// TwinCAT 3 PLC project SequentialTestSuitesAndTests
// Title: TcUnit sequentially running tests example projects
// Company: www.tcunit.org
// Author: Jakob Sagatowski
// ProjectVersion: 1.0.0.0
// ProgramVersion: 3.1.4022.7
// libraries:
//   Tc2_EtherCAT, * (Beckhoff Automation GmbH)
//   Tc2_Standard, * (Beckhoff Automation GmbH)
//   Tc2_System, * (Beckhoff Automation GmbH)
//   Tc3_Module, * (Beckhoff Automation GmbH)
//   TcUnit, * (www.tcunit.org)
// project tree:
//   DUTs/ E_DIAGNOSISTYPE.TcDUT, E_DIAGNOSTICCODETYPE.TcDUT, E_EVENTQUALIFIERMODE.TcDUT, E_TIMESTAMPTYPE.TcDUT (not stored), ST_DIAGNOSTICCODE.TcDUT (not stored), ST_DIAGNOSTICMESSAGE.TcDUT (not stored), ST_FLAGS.TcDUT (not stored)
//   GVLs/ GVL.TcGVL
//   / PlcTask.TcTTO
//   POUs/ FB_DiagnosticMessageDiagnosticCodeParser.TcPOU, FB_DiagnosticMessageFlagsParser.TcPOU, FB_DiagnosticMessageParser.TcPOU, FB_DiagnosticMessageTextIdentityParser.TcPOU, FB_DiagnosticMessageTimeStampParser.TcPOU, F_DWORDFromBytes.TcPOU (not stored), F_WORDFromBytes.TcPOU
//   Test/ FB_DiagnosticMessageDiagnosticCodeParser_Test.TcPOU, FB_DiagnosticMessageFlagsParser_Test.TcPOU, FB_DiagnosticMessageParser_Test.TcPOU, FB_DiagnosticMessageTextIdentityParser_Test.TcPOU, FB_DiagnosticMessageTimeStampParser_Test.TcPOU, PRG_TEST.TcPOU
// real-time tasks:
//   TASK PlcTask: cycle T#10ms, priority 20, ADS port 350

CONFIGURATION SequentialTestSuitesAndTests
    RESOURCE PLC ON TwinCAT3
        TASK PlcTask(INTERVAL := T#10ms, PRIORITY := 20);
        PROGRAM PRG_TEST WITH PlcTask : PRG_TEST;
    END_RESOURCE
END_CONFIGURATION

// ---- DUTs/E_DIAGNOSISTYPE.TcDUT
{attribute 'qualified_only'}
TYPE E_DIAGNOSISTYPE :
(
    InfoMessage := 0,
    WarningMessage := 1,
    ErrorMessage := 2,
    Unspecified := 3
) BYTE;
END_TYPE

// ---- DUTs/E_DIAGNOSTICCODETYPE.TcDUT
{attribute 'qualified_only'}
{attribute 'strict'}
TYPE E_DIAGNOSTICCODETYPE :
(
    ManufacturerSpecific := 0,
    EmergencyErrorCodeDS301 := 1,
    ProfileSpecific := 2,
    Unspecified := 3
) USINT;
END_TYPE

// ---- DUTs/E_EVENTQUALIFIERMODE.TcDUT
{attribute 'qualified_only'}
TYPE E_EVENTQUALIFIERMODE :
(
	Reserved := 0,
    EventSingleShot := 1,
    EventDisappears := 2,
    EventAppears := 3
) USINT;
END_TYPE

// ---- GVLs/GVL.TcGVL
{attribute 'qualified_only'}
VAR_GLOBAL
    fbDiagnosticMessageDiagnosticCodeParser_Test_WhenEmergencyErrorCodeExpectEmergencyErrorCode : ULINT;
    fbDiagnosticMessageDiagnosticCodeParser_Test_WhenManufacturerSpecificExpectManufacturerSpecific : ULINT;
    fbDiagnosticMessageDiagnosticCodeParser_Test_WhenProfileSpecificExpectProfileSpecific : ULINT;
    fbDiagnosticMessageDiagnosticCodeParser_Test_WhenReservedForFutureUseExpectReservedForFutureUse : ULINT;

    fbDiagnosticMessageFlagsParser_Test_WhenInfoMessageExpectInfoMessageGlobalTimestampAndZeroParameters : ULINT;
    fbDiagnosticMessageFlagsParser_Test_WhenWarningMessageExpectWarningMessageLocalTimestampAndTwoParameters : ULINT;
    fbDiagnosticMessageFlagsParser_Test_WhenErrorMessageExpectErrorMessageLocalTimestampAndFourParameters : ULINT;
    fbDiagnosticMessageFlagsParser_Test_WhenReservedForFutureUseMessageExpectReservedForFutureUseMessageLocalTimestampAnd33Parameters : ULINT;    

    fbDiagnosticMessageParser_Test_TestWithEmergencyMessage : ULINT;
    fbDiagnosticMessageParser_Test_TestWithManufacturerSpecificMessage : ULINT;
    fbDiagnosticMessageParser_Test_TestWithUnspecifiedMessageMessage : ULINT;
    fbDiagnosticMessageParser_Test_TestWithUnspecifiedMessageMessage_ParameterVariant : ULINT;

    fbDiagnosticMessageTextIdentityParser_Test_WhenTextIdentityLowExpectTextIdentity0 : ULINT;
    fbDiagnosticMessageTextIdentityParser_Test_WhenTextIdentityHighExpectTextIdentity65535 : ULINT;
    fbDiagnosticMessageTextIdentityParser_Test_WhenTextIdentityMedExpectTextIdentity34500 : ULINT;

    fbDiagnosticMessageTimeStampParser_Test_TestWithTimestampZeroTimeExpectCurrentTime : ULINT;
    fbDiagnosticMessageTimeStampParser_Test_TestWithValidTimestampExpectSameTimestamp : ULINT;
END_VAR

// ---- Test/PRG_TEST.TcPOU
(*
    This is the main program for execution of the unit tests.
    The program executes the test suites one after the other, with a delay of T#0MS between
    each other (that is, as soon as one test suite has finished executing, the next
    one starts to execute immediately after). This delay is defined in the parameter
    GVL_Param_TcUnit.TimeBetweenTestSuitesExecution (default T#0MS).
    Within each test suite, the program also executes each test one after the other, which
    is achieved by calling the TEST_ORDERED() for every test. The test-order is defined
    by the order of which the tests are being called.
*)
PROGRAM PRG_TEST
VAR
    (* Test function blocks *)
    fbDiagnosticMessageDiagnosticCodeParser_Test : FB_DiagnosticMessageDiagnosticCodeParser_Test;
    fbDiagnosticMessageFlagsParser_Test : FB_DiagnosticMessageFlagsParser_Test;
    fbDiagnosticMessageParser_Test : FB_DiagnosticMessageParser_Test;
    fbDiagnosticMessageTextIdentityParser_Test : FB_DiagnosticMessageTextIdentityParser_Test;
    fbDiagnosticMessageTimeStampParser_Test : FB_DiagnosticMessageTimeStampParser_Test;
END_VAR

TcUnit.RUN_IN_SEQUENCE();

END_PROGRAM

// ---- Test/FB_DiagnosticMessageDiagnosticCodeParser_Test.TcPOU
FUNCTION_BLOCK FB_DiagnosticMessageDiagnosticCodeParser_Test EXTENDS TcUnit.FB_TestSuite

(* The tests are run in the order that they are called. Asserts are not evaluated before the previous test has called TEST_FINISHED() *)
WhenEmergencyErrorCodeExpectEmergencyErrorCode();
WhenManufacturerSpecificExpectManufacturerSpecific();
WhenProfileSpecificExpectProfileSpecific();
WhenReservedForFutureUseExpectReservedForFutureUse();

METHOD PRIVATE WhenEmergencyErrorCodeExpectEmergencyErrorCode
VAR
    fbDiagnosticMessageDiagnosticCodeParser : FB_DiagnosticMessageDiagnosticCodeParser;
    stDiagnosticCode : ST_DIAGNOSTICCODE;
END_VAR
VAR CONSTANT
    // @TEST-FIXTURE EmergencyErrorCode
    cnDiagnosticCodeBufferByte1_EmergencyErrorCode : BYTE := 16#00; // 16#E800
    cnDiagnosticCodeBufferByte2_EmergencyErrorCode : BYTE := 16#E8;
    cnDiagnosticCodeBufferByte3_EmergencyErrorCode : BYTE := 16#30; // 16#7530 = 10#30000
    cnDiagnosticCodeBufferByte4_EmergencyErrorCode : BYTE := 16#75;
    canDiagnosticCodeBuffer_EmergencyErrorCode : ARRAY[1..4] OF BYTE := [
                                                cnDiagnosticCodeBufferByte1_EmergencyErrorCode,
                                                cnDiagnosticCodeBufferByte2_EmergencyErrorCode,
                                                cnDiagnosticCodeBufferByte3_EmergencyErrorCode,
                                                cnDiagnosticCodeBufferByte4_EmergencyErrorCode];
    // @TEST-RESULT EmergencyErrorCode
    ceDiagnosticCodeType_EmergencyErrorCode : E_DIAGNOSTICCODETYPE := E_DIAGNOSTICCODETYPE.EmergencyErrorCodeDS301;
    cnDiagnosticCode_EmergencyErrorCode : UINT := 10#30000;
END_VAR
IF TEST_ORDERED('WhenEmergencyErrorCodeExpectEmergencyErrorCode') THEN
    GVL.fbDiagnosticMessageDiagnosticCodeParser_Test_WhenEmergencyErrorCodeExpectEmergencyErrorCode := GVL.fbDiagnosticMessageDiagnosticCodeParser_Test_WhenEmergencyErrorCodeExpectEmergencyErrorCode + 1; // Only for testing the framework. Ignore this.
    // @TEST-RUN
    fbDiagnosticMessageDiagnosticCodeParser(anDiagnosticCodeBuffer := canDiagnosticCodeBuffer_EmergencyErrorCode,
                                            stDiagnosticCode => stDiagnosticCode);

    // @TEST-ASSERT
    AssertEquals_USINT(Expected := ceDiagnosticCodeType_EmergencyErrorCode,
                       Actual := stDiagnosticCode.eDiagnosticCodeType,
                       Message := 'Test $'emergency error code$' failed at $'diagnostic code type$'');
    AssertEquals_UINT(Expected := cnDiagnosticCode_EmergencyErrorCode,
                      Actual := stDiagnosticCode.nCode,
                      Message := 'Test $'emergency error code$' failed at $'diagnostic code$'');
    TEST_FINISHED();
END_IF
END_METHOD

METHOD PRIVATE WhenManufacturerSpecificExpectManufacturerSpecific
VAR
    fbDiagnosticMessageDiagnosticCodeParser : FB_DiagnosticMessageDiagnosticCodeParser;
    stDiagnosticCode : ST_DIAGNOSTICCODE;
END_VAR
VAR CONSTANT
    // @TEST-FIXTURE ManuFacturerSpecific
    cnDiagnosticCodeBufferByte1_ManufacturerSpecific : BYTE := 16#00; // 16#E000 (in range of 0xE000 - 0xE7FF)
    cnDiagnosticCodeBufferByte2_ManufacturerSpecific : BYTE := 16#E0;
    cnDiagnosticCodeBufferByte3_ManufacturerSpecific : BYTE := 16#E8; // 16#03E8 = 10#1000
    cnDiagnosticCodeBufferByte4_ManufacturerSpecific : BYTE := 16#03;
    canDiagnosticCodeBuffer_ManufacturerSpecific : ARRAY[1..4] OF BYTE := [
                                                cnDiagnosticCodeBufferByte1_ManufacturerSpecific,
                                                cnDiagnosticCodeBufferByte2_ManufacturerSpecific,
                                                cnDiagnosticCodeBufferByte3_ManufacturerSpecific,
                                                cnDiagnosticCodeBufferByte4_ManufacturerSpecific];
                                                
    // @TEST-RESULT ManuFacturerSpecific
    ceDiagnosticCodeType_ManufacturerSpecific : E_DIAGNOSTICCODETYPE := E_DIAGNOSTICCODETYPE.ManufacturerSpecific;
    cnDiagnosticCode_ManufacturerSpecific : UINT := 10#1000;
END_VAR
IF TEST_ORDERED('WhenManufacturerSpecificExpectManufacturerSpecific') THEN
    GVL.fbDiagnosticMessageDiagnosticCodeParser_Test_WhenManufacturerSpecificExpectManufacturerSpecific := GVL.fbDiagnosticMessageDiagnosticCodeParser_Test_WhenManufacturerSpecificExpectManufacturerSpecific + 1; // Only for testing the framework. Ignore this.
    // @TEST-RUN
    fbDiagnosticMessageDiagnosticCodeParser(anDiagnosticCodeBuffer := canDiagnosticCodeBuffer_ManufacturerSpecific,
                                            stDiagnosticCode => stDiagnosticCode);

    // @TEST-ASSERT
    AssertEquals_USINT(Expected := ceDiagnosticCodeType_ManufacturerSpecific,
                       Actual := stDiagnosticCode.eDiagnosticCodeType,
                       Message := 'Test $'manufacturer specific$' failed at $'diagnostic code type$'');
    AssertEquals_UINT(Expected := cnDiagnosticCode_ManufacturerSpecific,
                      Actual := stDiagnosticCode.nCode,
                      Message := 'Test $'manufacturer specific$' failed at $'diagnostic code$'');

    TEST_FINISHED();
END_IF
END_METHOD

METHOD PRIVATE WhenProfileSpecificExpectProfileSpecific
VAR
    fbDiagnosticMessageDiagnosticCodeParser : FB_DiagnosticMessageDiagnosticCodeParser;
    stDiagnosticCode : ST_DIAGNOSTICCODE;
END_VAR
VAR CONSTANT
    // @TEST-FIXTURE ProfileSpecific
    cnDiagnosticCodeBufferByte1_ProfileSpecific : BYTE := 16#10; // 16#EF10 (in range of 0xEE00 - 0xEFFF)
    cnDiagnosticCodeBufferByte2_ProfileSpecific : BYTE := 16#EF;
    cnDiagnosticCodeBufferByte3_ProfileSpecific : BYTE := 16#FF; // 16#FFFF = 10#65535
    cnDiagnosticCodeBufferByte4_ProfileSpecific : BYTE := 16#FF;
    canDiagnosticCodeBuffer_ProfileSpecific : ARRAY[1..4] OF BYTE := [
                                                cnDiagnosticCodeBufferByte1_ProfileSpecific,
                                                cnDiagnosticCodeBufferByte2_ProfileSpecific,
                                                cnDiagnosticCodeBufferByte3_ProfileSpecific,
                                                cnDiagnosticCodeBufferByte4_ProfileSpecific];

    // @TEST-RESULT ProfileSpecific
    ceDiagnosticCodeType_ProfileSpecific : E_DIAGNOSTICCODETYPE := E_DIAGNOSTICCODETYPE.ProfileSpecific;
    cnDiagnosticCode_ProfileSpecific : UINT := 10#65535;
END_VAR
IF TEST_ORDERED('WhenProfileSpecificExpectProfileSpecific') THEN
    GVL.fbDiagnosticMessageDiagnosticCodeParser_Test_WhenProfileSpecificExpectProfileSpecific := GVL.fbDiagnosticMessageDiagnosticCodeParser_Test_WhenProfileSpecificExpectProfileSpecific + 1; // Only for testing the framework. Ignore this.
    // @TEST-RUN
    fbDiagnosticMessageDiagnosticCodeParser(anDiagnosticCodeBuffer := canDiagnosticCodeBuffer_ProfileSpecific,
                                            stDiagnosticCode => stDiagnosticCode);

    // @TEST-ASSERT
    AssertEquals_USINT(Expected := ceDiagnosticCodeType_ProfileSpecific,
                       Actual := stDiagnosticCode.eDiagnosticCodeType,
                       Message := 'Test $'profile specific$' failed at $'diagnostic code type$'');
    AssertEquals_UINT(Expected := cnDiagnosticCode_ProfileSpecific,
                      Actual := stDiagnosticCode.nCode,
                      Message := 'Test $'profile specific$' failed at $'diagnostic code$'');

    TEST_FINISHED();
END_IF
END_METHOD

METHOD PRIVATE WhenReservedForFutureUseExpectReservedForFutureUse
VAR
    fbDiagnosticMessageDiagnosticCodeParser : FB_DiagnosticMessageDiagnosticCodeParser;
    stDiagnosticCode : ST_DIAGNOSTICCODE;
END_VAR
VAR CONSTANT
    // @TEST-FIXTURE ReservedForFutureUse
    cnDiagnosticCodeBufferByte1_ReservedForFutureUse : BYTE := 16#01; // 16#E801 (in range of 0xE801 - 0xEDFF)
    cnDiagnosticCodeBufferByte2_ReservedForFutureUse : BYTE := 16#E8;
    cnDiagnosticCodeBufferByte3_ReservedForFutureUse : BYTE := 16#D9; // 16#3BD9 = 10#15321
    cnDiagnosticCodeBufferByte4_ReservedForFutureUse : BYTE := 16#3B;
    canDiagnosticCodeBuffer_ReservedForFutureUse : ARRAY[1..4] OF BYTE := [
                                                cnDiagnosticCodeBufferByte1_ReservedForFutureUse,
                                                cnDiagnosticCodeBufferByte2_ReservedForFutureUse,
                                                cnDiagnosticCodeBufferByte3_ReservedForFutureUse,
                                                cnDiagnosticCodeBufferByte4_ReservedForFutureUse];

    // @TEST-RESULT ReservedForFutureUse
    ceDiagnosticCodeType_ReservedForFutureUse : E_DIAGNOSTICCODETYPE := E_DIAGNOSTICCODETYPE.Unspecified;
    cnDiagnosticCode_ReservedForFutureUse : UINT := 10#15321;
END_VAR
IF TEST_ORDERED('WhenReservedForFutureUseExpectReservedForFutureUse') THEN
    GVL.fbDiagnosticMessageDiagnosticCodeParser_Test_WhenReservedForFutureUseExpectReservedForFutureUse := GVL.fbDiagnosticMessageDiagnosticCodeParser_Test_WhenReservedForFutureUseExpectReservedForFutureUse + 1; // Only for testing the framework. Ignore this.

    // @TEST-RUN
    fbDiagnosticMessageDiagnosticCodeParser(anDiagnosticCodeBuffer := canDiagnosticCodeBuffer_ReservedForFutureUse,
                                            stDiagnosticCode => stDiagnosticCode);

    // @TEST-ASSERT
    AssertEquals_USINT(Expected := ceDiagnosticCodeType_ReservedForFutureUse,
                       Actual := stDiagnosticCode.eDiagnosticCodeType,
                       Message := 'Test $'reserved for future use$' failed at $'diagnostic code type$'');
    AssertEquals_UINT(Expected := cnDiagnosticCode_ReservedForFutureUse,
                      Actual := stDiagnosticCode.nCode,
                      Message := 'Test $'reserved for future use$' failed at $'diagnostic code$'');

    TEST_FINISHED();
END_IF
END_METHOD

END_FUNCTION_BLOCK

// ---- POUs/FB_DiagnosticMessageDiagnosticCodeParser.TcPOU
(*
    This function block parses a the part "diagnostic code" of the diagnostic message according to the
    ETG.1020 protocol enhancements.
*)
FUNCTION_BLOCK FB_DiagnosticMessageDiagnosticCodeParser
VAR_INPUT
    anDiagnosticCodeBuffer : ARRAY[1..4] OF BYTE;
END_VAR
VAR_OUTPUT
    stDiagnosticCode : ST_DIAGNOSTICCODE;
END_VAR
VAR
    nDiagnosisCodeType : WORD;
    nDiagnosisCodeTypeLow : WORD;
    nCode : WORD;
    nCodeLow : WORD;
END_VAR
VAR CONSTANT
    cnNotUsedOne_Low : WORD := 16#0000;
    cnNotUsedOne_High : WORD := 16#DFFF;
    cnManufacturerSpecific_Low : WORD := 16#E000;
    cnManufacturerSpecific_High : WORD := 16#E7FF;
    cnEmergencyErrorCodeDS301 : WORD := 16#E800;
    cnReservedForFutureStandardization_Low : WORD := 16#E801;
    cnReservedForFutureStandardization_High : WORD := 16#EDFF;
    cnProfileSpecific_Low : WORD := 16#EE00;
    cnProfileSpecific_High : WORD := 16#EFFF;
    cnNotUsedTwo_Low : WORD := 16#F000;
    cnNotUsedTwo_High : WORD := 16#FFFF;
END_VAR

nDiagnosisCodeType := BYTE_TO_WORD(anDiagnosticCodeBuffer[2]);
nDiagnosisCodeType := SHL(nDiagnosisCodeType, 8);
nDiagnosisCodeTypeLow := BYTE_TO_WORD(anDiagnosticCodeBuffer[1]);
nDiagnosisCodeType := nDiagnosisCodeType OR nDiagnosisCodeTypeLow;

IF (nDiagnosisCodeType >= cnNotUsedOne_Low AND nDiagnosisCodeType <= cnNotUsedOne_High) OR
   (nDiagnosisCodeType >= cnReservedForFutureStandardization_Low AND
    nDiagnosisCodeType <= cnReservedForFutureStandardization_High) OR
   (nDiagnosisCodeType >= cnNotUsedTwo_Low AND nDiagnosisCodeType <= cnNotUsedTwo_High) THEN
   stDiagnosticCode.eDiagnosticCodeType := E_DIAGNOSTICCODETYPE.Unspecified;
ELSIF nDiagnosisCodeType >= cnManufacturerSpecific_Low AND nDiagnosisCodeType <= cnManufacturerSpecific_High THEN
    stDiagnosticCode.eDiagnosticCodeType := E_DIAGNOSTICCODETYPE.ManufacturerSpecific;
ELSIF nDiagnosisCodeType = cnEmergencyErrorCodeDS301 THEN
    stDiagnosticCode.eDiagnosticCodeType := E_DIAGNOSTICCODETYPE.EmergencyErrorCodeDS301;
ELSIF nDiagnosisCodeType >= cnProfileSpecific_Low AND nDiagnosisCodeType <= cnProfileSpecific_High THEN
    stDiagnosticCode.eDiagnosticCodeType := E_DIAGNOSTICCODETYPE.ProfileSpecific;
END_IF

nCode := BYTE_TO_WORD(anDiagnosticCodeBuffer[4]);
nCode := SHL(nCode, 8);
nCodeLow := BYTE_TO_WORD(anDiagnosticCodeBuffer[3]);
nCode := nCode OR nCodeLow;

stDiagnosticCode.nCode := WORD_TO_UINT(nCode);

END_FUNCTION_BLOCK

// ---- Test/FB_DiagnosticMessageFlagsParser_Test.TcPOU
FUNCTION_BLOCK FB_DiagnosticMessageFlagsParser_Test EXTENDS TcUnit.FB_TestSuite

(* The tests are run in the order that they are called. Asserts are not evaluated before the previous test has called TEST_FINISHED() *)
WhenInfoMessageExpectInfoMessageGlobalTimestampAndZeroParameters();
WhenWarningMessageExpectWarningMessageLocalTimestampAndTwoParameters();
WhenErrorMessageExpectErrorMessageLocalTimestampAndFourParameters();
WhenReservedForFutureUseMessageExpectReservedForFutureUseMessageLocalTimestampAnd33Parameters();

METHOD PRIVATE WhenErrorMessageExpectErrorMessageLocalTimestampAndFourParameters
VAR
    fbDiagnosticMessageFlagsParser : FB_DiagnosticMessageFlagsParser;
    stFlags : ST_FLAGS;

    // @TEST-FIXTURE ErrorMessage
    cnFlagsBufferByte1_ErrorMessage : BYTE := 2#0001_0010; // Error message and local time stamp
    cnFlagsBufferByte2_ErrorMessage : BYTE := 2#0000_0100; // Four parameters in the diagnosis message
    canFlagsBuffer_ErrorMessage : ARRAY[1..2] OF BYTE := [cnFlagsBufferByte1_ErrorMessage, 
                                                          cnFlagsBufferByte2_ErrorMessage];
    // @TEST-RESULT ErrorMessage
    ceFlags_DiagnosisTypeErrorMessage : E_DIAGNOSISTYPE := E_DIAGNOSISTYPE.ErrorMessage;
    ceFlags_TimeStampTypeLocal : E_TIMESTAMPTYPE := E_TIMESTAMPTYPE.Local;
    cnFlags_NumberOfParametersInDiagnosisMessageFour : USINT := 4;
END_VAR
IF TEST_ORDERED('WhenErrorMessageExpectErrorMessageLocalTimestampAndFourParameters') THEN
    GVL.fbDiagnosticMessageFlagsParser_Test_WhenErrorMessageExpectErrorMessageLocalTimestampAndFourParameters := GVL.fbDiagnosticMessageFlagsParser_Test_WhenErrorMessageExpectErrorMessageLocalTimestampAndFourParameters + 1; // Only for testing the framework. Ignore this.

    // @TEST-RUN ErrorMessage
    fbDiagnosticMessageFlagsParser(anFlagsBuffer := canFlagsBuffer_ErrorMessage,
                                   stFlags => stFlags);

    // @TEST-ASSERT ErrorMessage
    AssertEquals(Expected := ceFlags_DiagnosisTypeErrorMessage,
                 Actual := stFlags.eDiagnosisType,
                 'Test $'Error message$' failed at $'diagnosis type$'');
    AssertEquals(Expected := ceFlags_TimeStampTypeLocal,
                 Actual := stFlags.eTimeStampType,
                 'Test $'Error message$' failed at $'timestamp type$'');
    AssertEquals(Expected := cnFlags_NumberOfParametersInDiagnosisMessageFour,
                 Actual := stFlags.nNumberOfParametersInDiagnosisMessage,
                 'Test $'Error message$' failed at $'number of parameters$'');

    TEST_FINISHED();
END_IF
END_METHOD

METHOD PRIVATE WhenInfoMessageExpectInfoMessageGlobalTimestampAndZeroParameters
VAR
    fbDiagnosticMessageFlagsParser : FB_DiagnosticMessageFlagsParser;
    stFlags : ST_FLAGS;

    // @TEST-FIXTURE InfoMessage
    cnFlagsBufferByte1_InfoMessage : BYTE := 2#0000_0000; // Info message and global time stamp
    cnFlagsBufferByte2_InfoMessage : BYTE := 2#0000_0000; // Zero parameters in the diagnosis message
    canFlagsBuffer_InfoMessage : ARRAY[1..2] OF BYTE := [cnFlagsBufferByte1_InfoMessage, 
                                                         cnFlagsBufferByte2_InfoMessage];
    // @TEST-RESULT InfoMessage
    ceFlags_DiagnosisTypeInfoMessage : E_DIAGNOSISTYPE := E_DIAGNOSISTYPE.InfoMessage;
    ceFlags_TimeStampTypeGlobal : E_TIMESTAMPTYPE := E_TIMESTAMPTYPE.Global;
    cnFlags_NumberOfParametersInDiagnosisMessageZero : USINT := 0;
END_VAR
IF TEST_ORDERED('WhenInfoMessageExpectInfoMessageGlobalTimestampAndZeroParameters') THEN
    GVL.fbDiagnosticMessageFlagsParser_Test_WhenInfoMessageExpectInfoMessageGlobalTimestampAndZeroParameters := GVL.fbDiagnosticMessageFlagsParser_Test_WhenInfoMessageExpectInfoMessageGlobalTimestampAndZeroParameters + 1; // Only for testing the framework. Ignore this.

    // @TEST-RUN
    fbDiagnosticMessageFlagsParser(anFlagsBuffer := canFlagsBuffer_InfoMessage,
                                   stFlags => stFlags);

    // @TEST-ASSERT
    AssertEquals(Expected := ceFlags_DiagnosisTypeInfoMessage,
                 Actual := stFlags.eDiagnosisType,
                 'Test $'Info message$' failed at $'diagnosis type$'');
    AssertEquals(Expected := ceFlags_TimeStampTypeGlobal,
                 Actual := stFlags.eTimeStampType,
                 'Test $'Info message$' failed at $'timestamp type$'');
    AssertEquals(Expected := cnFlags_NumberOfParametersInDiagnosisMessageZero,
                 Actual := stFlags.nNumberOfParametersInDiagnosisMessage,
                 'Test $'Info message$' failed at $'number of parameters$'');

    TEST_FINISHED();
END_IF
END_METHOD

METHOD PRIVATE WhenReservedForFutureUseMessageExpectReservedForFutureUseMessageLocalTimestampAnd33Parameters
VAR
    fbDiagnosticMessageFlagsParser : FB_DiagnosticMessageFlagsParser;
    stFlags : ST_FLAGS;

    // @TEST-FIXTURE ReservedForFutureUseMessage
    cnFlagsBufferByte1_ReservedForFutureUseMessage : BYTE := 2#0001_0011; // ReservedForFutureUse message and local time stamp
    cnFlagsBufferByte2_ReservedForFutureUseMessage : BYTE := 2#0010_0001; // 33 parameters in the diagnosis message
    canFlagsBuffer_ReservedForFutureUseMessage : ARRAY[1..2] OF BYTE := [cnFlagsBufferByte1_ReservedForFutureUseMessage, 
                                                                         cnFlagsBufferByte2_ReservedForFutureUseMessage];
    // @TEST-RESULT ReservedForFutureUseMessage
    ceFlags_DiagnosisTypeReservedForFutureUseMessage : E_DIAGNOSISTYPE := E_DIAGNOSISTYPE.Unspecified;
    cnFlags_NumberOfParametersInDiagnosisMessage33 : USINT := 33;
    ceFlags_TimeStampTypeLocal : E_TIMESTAMPTYPE := E_TIMESTAMPTYPE.Local;
END_VAR
IF TEST_ORDERED('WhenReservedForFutureUseMessageExpectReservedForFutureUseMessageLocalTimestampAnd33Parameters') THEN
    GVL.fbDiagnosticMessageFlagsParser_Test_WhenReservedForFutureUseMessageExpectReservedForFutureUseMessageLocalTimestampAnd33Parameters := GVL.fbDiagnosticMessageFlagsParser_Test_WhenReservedForFutureUseMessageExpectReservedForFutureUseMessageLocalTimestampAnd33Parameters + 1; // Only for testing the framework. Ignore this.

    // @TEST-RUN ReservedForFutureUseMessage
    fbDiagnosticMessageFlagsParser(anFlagsBuffer := canFlagsBuffer_ReservedForFutureUseMessage,
                                   stFlags => stFlags);

    // @TEST-ASSERT ReservedForFutureUseMessage
    AssertEquals(Expected := ceFlags_DiagnosisTypeReservedForFutureUseMessage,
                 Actual := stFlags.eDiagnosisType,
                 'Test $'Reserved for future use message$' failed at $'diagnosis type$'');
    AssertEquals(Expected := ceFlags_TimeStampTypeLocal,
                 Actual := stFlags.eTimeStampType,
                 'Test $'Reserved for future use message$' failed at $'timestamp type$'');
    AssertEquals(Expected := cnFlags_NumberOfParametersInDiagnosisMessage33,
                 Actual := stFlags.nNumberOfParametersInDiagnosisMessage,
                 'Test $'Reserved for future use message$' failed at $'number of parameters$'');

    TEST_FINISHED();
END_IF
END_METHOD

METHOD PRIVATE WhenWarningMessageExpectWarningMessageLocalTimestampAndTwoParameters
VAR
    fbDiagnosticMessageFlagsParser : FB_DiagnosticMessageFlagsParser;
    stFlags : ST_FLAGS;

    // @TEST-FIXTURE WarningMessage
    cnFlagsBufferByte1_WarningMessage : BYTE := 2#0001_0001; // Warning message and local time stamp
    cnFlagsBufferByte2_WarningMessage : BYTE := 2#0000_0010; // Two parameters in the diagnosis message
    canFlagsBuffer_WarningMessage : ARRAY[1..2] OF BYTE := [cnFlagsBufferByte1_WarningMessage, 
                                                            cnFlagsBufferByte2_WarningMessage];
    // @TEST-RESULT WarningMessage
    ceFlags_DiagnosisTypeWarningMessage : E_DIAGNOSISTYPE := E_DIAGNOSISTYPE.WarningMessage;
    ceFlags_TimeStampTypeLocal : E_TIMESTAMPTYPE := E_TIMESTAMPTYPE.Local;
    cnFlags_NumberOfParametersInDiagnosisMessageTwo : USINT := 2;
END_VAR
IF TEST_ORDERED('WhenWarningMessageExpectWarningMessageLocalTimestampAndTwoParameters') THEN
    GVL.fbDiagnosticMessageFlagsParser_Test_WhenWarningMessageExpectWarningMessageLocalTimestampAndTwoParameters := GVL.fbDiagnosticMessageFlagsParser_Test_WhenWarningMessageExpectWarningMessageLocalTimestampAndTwoParameters + 1; // Only for testing the framework. Ignore this.

    // @TEST-RUN WarningMessage
    fbDiagnosticMessageFlagsParser(anFlagsBuffer := canFlagsBuffer_WarningMessage,
                                   stFlags => stFlags);

    // @TEST-ASSERT WarningMessage
    AssertEquals(Expected := ceFlags_DiagnosisTypeWarningMessage,
                 Actual := stFlags.eDiagnosisType,
                 'Test $'Warning message$' failed at $'diagnosis type$'');
    AssertEquals(Expected := ceFlags_TimeStampTypeLocal,
                 Actual := stFlags.eTimeStampType,
                 'Test $'Warning message$' failed at $'timestamp type$'');
    AssertEquals(Expected := cnFlags_NumberOfParametersInDiagnosisMessageTwo,
                 Actual := stFlags.nNumberOfParametersInDiagnosisMessage,
                 'Test $'Warning message$' failed at $'number of parameters$'');

    TEST_FINISHED();

END_IF
END_METHOD

END_FUNCTION_BLOCK

// ---- POUs/FB_DiagnosticMessageFlagsParser.TcPOU
(*
    This function block parses a the part "flags" of the diagnostic message according to the
    ETG.1020 protocol enhancements.
*)
FUNCTION_BLOCK FB_DiagnosticMessageFlagsParser
VAR_INPUT
    anFlagsBuffer : ARRAY[1..2] OF BYTE;
END_VAR
VAR_OUTPUT
    stFlags : ST_FLAGS;
END_VAR
VAR
    nFlags : BYTE;
END_VAR

nFlags.0 := anFlagsBuffer[1].0;
nFlags.1 := anFlagsBuffer[1].1;
nFlags.2 := anFlagsBuffer[1].2;
nFlags.3 := anFlagsBuffer[1].3;

IF nFlags >= 10#0 AND nFlags <= 10#2 THEN
    stFlags.eDiagnosisType := nFlags;
ELSE
    stFlags.eDiagnosisType := E_DIAGNOSISTYPE.Unspecified;
END_IF

IF anFlagsBuffer[1].4 THEN
    stFlags.eTimeStampType := E_TIMESTAMPTYPE.Local;
ELSE
    stFlags.eTimeStampType := E_TIMESTAMPTYPE.Global;
END_IF

stFlags.nNumberOfParametersInDiagnosisMessage := BYTE_TO_USINT(anFlagsBuffer[2]);

END_FUNCTION_BLOCK

// ---- Test/FB_DiagnosticMessageParser_Test.TcPOU
FUNCTION_BLOCK FB_DiagnosticMessageParser_Test EXTENDS TcUnit.FB_TestSuite

(* The tests are run in the order that they are called. Asserts are not evaluated before the previous test has called TEST_FINISHED() *)
TestWithEmergencyMessage();
TestWithManufacturerSpecificMessage();
TestWithUnspecifiedMessageMessage();
TestWithUnspecifiedMessageMessage_ParameterVariant();

METHOD PRIVATE TestWithEmergencyMessage
VAR  
    fbDiagnosticMessageParser : FB_DiagnosticMessageParser;
    aDiagnosticMessageBuffer : ARRAY[1..28] OF BYTE;
    stDiagnosticMessage : ST_DIAGNOSTICMESSAGE;

    // @TEST-RESULT EmergencyMessage
    stDiagnosticMessage_EmergencyMessage : ST_DIAGNOSTICMESSAGE :=
        (stDiagnosticCode := (eDiagnosticCodeType := E_DIAGNOSTICCODETYPE.EmergencyErrorCodeDS301, nCode := 0),
        stFlags := (eDiagnosisType := E_DIAGNOSISTYPE.ErrorMessage, eTimeStampType := E_TIMESTAMPTYPE.Local,
                    nNumberOfParametersInDiagnosisMessage := 0),
        nTextIdentityReferenceToESIFile := 0,
        sTimeStamp := '');  // Local time stamp, will be updated in program call to current task time;

    // @TEST-FIXTURE EmergencyMessage
    cnDiagnosticBufferByte1_EmergencyMessage : BYTE := 16#00; // 0xE800 = Emergency code
    cnDiagnosticBufferByte2_EmergencyMessage : BYTE := 16#E8;
    cnDiagnosticBufferByte3_EmergencyMessage : BYTE := 16#00; // 0x0000 = Code 0
    cnDiagnosticBufferByte4_EmergencyMessage : BYTE := 16#00;
    cnDiagnosticBufferByte5_EmergencyMessage : BYTE := 2#0001_0010; // Local time stamp & error message 
    cnDiagnosticBufferByte6_EmergencyMessage : BYTE := 16#00; // Number of parameters = 0
    cnDiagnosticBufferByte7_EmergencyMessage : BYTE := 16#00; // 0x0000, Text id as reference to ESI file = 0
    cnDiagnosticBufferByte8_EmergencyMessage : BYTE := 16#00;
    cnDiagnosticBufferByte9_16_EmergencyMessage : BYTE := 16#00; // Timestamp (none attached)
    cnDiagnosticBufferByte17_EmergencyMessage : BYTE := 2#0000_0010; // Param1 = Signed8
    cnDiagnosticBufferByte18_EmergencyMessage : BYTE := 2#0000_0000;
    cnDiagnosticBufferByte19_EmergencyMessage : BYTE := 2#0000_0011; // Port 3
    cnDiagnosticBufferByte20_EmergencyMessage : BYTE := 2#0000_0011; // Param2 = Signed16
    cnDiagnosticBufferByte21_EmergencyMessage : BYTE := 2#0000_0000;
    cnDiagnosticBufferByte22_EmergencyMessage : BYTE := 2#1110_1000; // EventCode = 10#1000
    cnDiagnosticBufferByte23_EmergencyMessage : BYTE := 2#0000_0011;
    cnDiagnosticBufferByte24_EmergencyMessage : BYTE := 2#0000_0010; // Param3 = Signed8
    cnDiagnosticBufferByte25_EmergencyMessage : BYTE := 2#0000_0000;
    cnDiagnosticBufferByte26_EmergencyMessage : BYTE := 2#0001_0111; // Qualifier: Instance=Reserved_7, Source=Device, Type=Notification, Mode=Reserved
    cnDiagnosticBufferByte27_EmergencyMessage : BYTE := 2#0000_0000;
    cnDiagnosticBufferByte28_EmergencyMessage : BYTE := 2#0000_0000;

    canDiagnosticBuffer_EmergencyMessage : ARRAY[1..28] OF BYTE := [cnDiagnosticBufferByte1_EmergencyMessage,
                                                                    cnDiagnosticBufferByte2_EmergencyMessage,
                                                                    cnDiagnosticBufferByte3_EmergencyMessage,
                                                                    cnDiagnosticBufferByte4_EmergencyMessage,
                                                                    cnDiagnosticBufferByte5_EmergencyMessage,
                                                                    cnDiagnosticBufferByte6_EmergencyMessage,
                                                                    cnDiagnosticBufferByte7_EmergencyMessage,
                                                                    cnDiagnosticBufferByte8_EmergencyMessage,
                                                                    8(cnDiagnosticBufferByte9_16_EmergencyMessage),
                                                                    cnDiagnosticBufferByte17_EmergencyMessage,
                                                                    cnDiagnosticBufferByte18_EmergencyMessage,
                                                                    cnDiagnosticBufferByte19_EmergencyMessage,
                                                                    cnDiagnosticBufferByte20_EmergencyMessage,
                                                                    cnDiagnosticBufferByte21_EmergencyMessage,
                                                                    cnDiagnosticBufferByte22_EmergencyMessage,
                                                                    cnDiagnosticBufferByte23_EmergencyMessage,
                                                                    cnDiagnosticBufferByte24_EmergencyMessage,
                                                                    cnDiagnosticBufferByte25_EmergencyMessage,
                                                                    cnDiagnosticBufferByte26_EmergencyMessage,
                                                                    cnDiagnosticBufferByte27_EmergencyMessage,
                                                                    cnDiagnosticBufferByte28_EmergencyMessage];
END_VAR
IF TEST_ORDERED('TestWithEmergencyMessage') THEN
    GVL.fbDiagnosticMessageParser_Test_TestWithEmergencyMessage := GVL.fbDiagnosticMessageParser_Test_TestWithEmergencyMessage + 1; // Only for testing the framework. Ignore this.

    // @TEST-RUN
    stDiagnosticMessage_EmergencyMessage.sTimeStamp := DCTIME64_TO_STRING(in := F_GetCurDcTaskTime64());

    fbDiagnosticMessageParser(anDiagnosticMessageBuffer := canDiagnosticBuffer_EmergencyMessage,
                              stDiagnosticMessage => stDiagnosticMessage);

    // @TEST-ASSERT
    AssertEquals(Expected := stDiagnosticMessage_EmergencyMessage.stDiagnosticCode.eDiagnosticCodeType,
                 Actual := stDiagnosticMessage.stDiagnosticCode.eDiagnosticCodeType,
                 Message := 'Test $'EmergencyMessage$' failed at $'Diagnostic code type$'');
    AssertEquals(Expected := stDiagnosticMessage_EmergencyMessage.stDiagnosticCode.nCode,
                 Actual := stDiagnosticMessage.stDiagnosticCode.nCode,
                 Message := 'Test $'EmergencyMessage$' failed at $'Diagnostic code$'');
    AssertEquals(Expected := stDiagnosticMessage_EmergencyMessage.stFlags.eDiagnosisType,
                 Actual := stDiagnosticMessage.stFlags.eDiagnosisType,
                 Message := 'Test $'EmergencyMessage$' failed at $'Diagnosis type$'');
    AssertEquals(Expected := stDiagnosticMessage_EmergencyMessage.stFlags.eTimeStampType,
                 Actual := stDiagnosticMessage.stFlags.eTimeStampType,
                 Message := 'Test $'EmergencyMessage$' failed at $'Timestamp type$'');
    AssertEquals(Expected := stDiagnosticMessage_EmergencyMessage.stFlags.nNumberOfParametersInDiagnosisMessage,
                 Actual := stDiagnosticMessage.stFlags.nNumberOfParametersInDiagnosisMessage,
                 Message := 'Test $'EmergencyMessage$' failed at $'Numbers of parameters in diagnosis message$'');
    AssertEquals(Expected := stDiagnosticMessage_EmergencyMessage.nTextIdentityReferenceToESIFile,
                 Actual := stDiagnosticMessage.nTextIdentityReferenceToESIFile,
                 Message := 'Test $'EmergencyMessage$' failed at $'Text identity reference to ESI file$'');
    AssertEquals(Expected := stDiagnosticMessage_EmergencyMessage.sTimeStamp,
                 Actual := stDiagnosticMessage.sTimeStamp,
                 Message := 'Test $'EmergencyMessage$' failed at $'Timestamp$'');

    TEST_FINISHED();
END_IF
END_METHOD

METHOD PRIVATE TestWithManufacturerSpecificMessage
VAR
    fbDiagnosticMessageParser : FB_DiagnosticMessageParser;
    aDiagnosticMessageBuffer : ARRAY[1..28] OF BYTE;
    stDiagnosticMessage : ST_DIAGNOSTICMESSAGE;

    // @TEST-FIXTURE ManufacturerSpecificMessage
    cnDiagnosticBufferByte1_ManufacturerSpecificMessage : BYTE := 16#90; // 0xE290 = Manufacturer Specific
    cnDiagnosticBufferByte2_ManufacturerSpecificMessage : BYTE := 16#E2;
    cnDiagnosticBufferByte3_ManufacturerSpecificMessage : BYTE := 16#30; // 0x0000 = Code 0
    cnDiagnosticBufferByte4_ManufacturerSpecificMessage : BYTE := 16#75;
    cnDiagnosticBufferByte5_ManufacturerSpecificMessage : BYTE := 2#0000_0000; // Global time stamp & info message 
    cnDiagnosticBufferByte6_ManufacturerSpecificMessage : BYTE := 16#02; // Number of parameters = 2
    cnDiagnosticBufferByte7_ManufacturerSpecificMessage : BYTE := 16#A8; // 0x61A8, Text id as reference to ESI file = 10#25000
    cnDiagnosticBufferByte8_ManufacturerSpecificMessage : BYTE := 16#61;
    cnDiagnosticBufferByte9_ManufacturerSpecificMessage : BYTE := 16#C8; // Timestamp from DC clock, 16#07C8D11492616FC8 = '2017-10-10-05:20:39.893037000'
    cnDiagnosticBufferByte10_ManufacturerSpecificMessage : BYTE := 16#6F;
    cnDiagnosticBufferByte11_ManufacturerSpecificMessage : BYTE := 16#61;
    cnDiagnosticBufferByte12_ManufacturerSpecificMessage : BYTE := 16#92;
    cnDiagnosticBufferByte13_ManufacturerSpecificMessage : BYTE := 16#14;
    cnDiagnosticBufferByte14_ManufacturerSpecificMessage : BYTE := 16#D1;
    cnDiagnosticBufferByte15_ManufacturerSpecificMessage : BYTE := 16#C8;
    cnDiagnosticBufferByte16_ManufacturerSpecificMessage : BYTE := 16#07;
    cnDiagnosticBufferByte17_ManufacturerSpecificMessage : BYTE := 2#0000_0010; // Param1 = Signed8
    cnDiagnosticBufferByte18_ManufacturerSpecificMessage : BYTE := 2#0000_0000;
    cnDiagnosticBufferByte19_ManufacturerSpecificMessage : BYTE := 2#0000_0110; // Port 6
    cnDiagnosticBufferByte20_ManufacturerSpecificMessage : BYTE := 2#0000_0011; // Param2 = Signed16
    cnDiagnosticBufferByte21_ManufacturerSpecificMessage : BYTE := 2#0000_0000;
    cnDiagnosticBufferByte22_ManufacturerSpecificMessage : BYTE := 2#1101_0010; // EventCode = 10#1234
    cnDiagnosticBufferByte23_ManufacturerSpecificMessage : BYTE := 2#0000_0100;
    cnDiagnosticBufferByte24_ManufacturerSpecificMessage : BYTE := 2#0000_0010; // Param3 = Signed8
    cnDiagnosticBufferByte25_ManufacturerSpecificMessage : BYTE := 2#0000_0000;
    cnDiagnosticBufferByte26_ManufacturerSpecificMessage : BYTE := 2#0100_0110; // Qualifier: Instance=Reserved_6, Source=Device, Type=Reserved, Mode=EventSingleShot
    cnDiagnosticBufferByte27_ManufacturerSpecificMessage : BYTE := 2#0000_0000;
    cnDiagnosticBufferByte28_ManufacturerSpecificMessage : BYTE := 2#0000_0000;

    canDiagnosticBuffer_ManufacturerSpecificMessage : ARRAY[1..28] OF BYTE := [
                                                               cnDiagnosticBufferByte1_ManufacturerSpecificMessage,
                                                               cnDiagnosticBufferByte2_ManufacturerSpecificMessage,
                                                               cnDiagnosticBufferByte3_ManufacturerSpecificMessage,
                                                               cnDiagnosticBufferByte4_ManufacturerSpecificMessage,
                                                               cnDiagnosticBufferByte5_ManufacturerSpecificMessage,
                                                               cnDiagnosticBufferByte6_ManufacturerSpecificMessage,
                                                               cnDiagnosticBufferByte7_ManufacturerSpecificMessage,
                                                               cnDiagnosticBufferByte8_ManufacturerSpecificMessage,
                                                               cnDiagnosticBufferByte9_ManufacturerSpecificMessage,
                                                               cnDiagnosticBufferByte10_ManufacturerSpecificMessage,
                                                               cnDiagnosticBufferByte11_ManufacturerSpecificMessage,
                                                               cnDiagnosticBufferByte12_ManufacturerSpecificMessage,
                                                               cnDiagnosticBufferByte13_ManufacturerSpecificMessage,
                                                               cnDiagnosticBufferByte14_ManufacturerSpecificMessage,
                                                               cnDiagnosticBufferByte15_ManufacturerSpecificMessage,
                                                               cnDiagnosticBufferByte16_ManufacturerSpecificMessage,
                                                               cnDiagnosticBufferByte17_ManufacturerSpecificMessage,
                                                               cnDiagnosticBufferByte18_ManufacturerSpecificMessage,
                                                               cnDiagnosticBufferByte19_ManufacturerSpecificMessage,
                                                               cnDiagnosticBufferByte20_ManufacturerSpecificMessage,
                                                               cnDiagnosticBufferByte21_ManufacturerSpecificMessage,
                                                               cnDiagnosticBufferByte22_ManufacturerSpecificMessage,
                                                               cnDiagnosticBufferByte23_ManufacturerSpecificMessage,
                                                               cnDiagnosticBufferByte24_ManufacturerSpecificMessage,
                                                               cnDiagnosticBufferByte25_ManufacturerSpecificMessage,
                                                               cnDiagnosticBufferByte26_ManufacturerSpecificMessage,
                                                               cnDiagnosticBufferByte27_ManufacturerSpecificMessage,
                                                               cnDiagnosticBufferByte28_ManufacturerSpecificMessage];

    // @TEST-RESULT ManufacturerSpecificMessage
    cstDiagnosticMessage_ManufacturerSpecificMessage : ST_DIAGNOSTICMESSAGE :=
        (stDiagnosticCode := (eDiagnosticCodeType := E_DIAGNOSTICCODETYPE.ManufacturerSpecific, nCode := 30000),
        stFlags := (eDiagnosisType := E_DIAGNOSISTYPE.InfoMessage, eTimeStampType := E_TIMESTAMPTYPE.Global,
                    nNumberOfParametersInDiagnosisMessage := 2),
        nTextIdentityReferenceToESIFile := 25000,
        sTimeStamp := '2017-10-10-05:20:39.893037000');
END_VAR
IF TEST_ORDERED('TestWithManufacturerSpecificMessage') THEN
    GVL.fbDiagnosticMessageParser_Test_TestWithManufacturerSpecificMessage := GVL.fbDiagnosticMessageParser_Test_TestWithManufacturerSpecificMessage + 1; // Only for testing the framework. Ignore this.

    // @TEST-RUN
    fbDiagnosticMessageParser(anDiagnosticMessageBuffer := canDiagnosticBuffer_ManufacturerSpecificMessage,
                              stDiagnosticMessage => stDiagnosticMessage);

    // @TEST-ASSERT
    AssertEquals(Expected := cstDiagnosticMessage_ManufacturerSpecificMessage.stDiagnosticCode.eDiagnosticCodeType,
                 Actual := stDiagnosticMessage.stDiagnosticCode.eDiagnosticCodeType,
                 Message := 'Test $'ManufacturerSpecificMessage$' failed at $'Diagnostic code type$'');
    AssertEquals(Expected := cstDiagnosticMessage_ManufacturerSpecificMessage.stDiagnosticCode.nCode,
                 Actual := stDiagnosticMessage.stDiagnosticCode.nCode,
                 Message := 'Test $'ManufacturerSpecificMessage$' failed at $'Diagnostic code$'');
    AssertEquals(Expected := cstDiagnosticMessage_ManufacturerSpecificMessage.stFlags.eDiagnosisType,
                 Actual := stDiagnosticMessage.stFlags.eDiagnosisType,
                 Message := 'Test $'ManufacturerSpecificMessage$' failed at $'Diagnosis type$'');
    AssertEquals(Expected := cstDiagnosticMessage_ManufacturerSpecificMessage.stFlags.eTimeStampType,
                 Actual := stDiagnosticMessage.stFlags.eTimeStampType,
                 Message := 'Test $'ManufacturerSpecificMessage$' failed at $'Timestamp type$'');
    AssertEquals(Expected := cstDiagnosticMessage_ManufacturerSpecificMessage.stFlags.nNumberOfParametersInDiagnosisMessage,
                 Actual := stDiagnosticMessage.stFlags.nNumberOfParametersInDiagnosisMessage,
                 Message := 'Test $'ManufacturerSpecificMessage$' failed at $'Numbers of parameters in diagnosis message$'');
    AssertEquals(Expected := cstDiagnosticMessage_ManufacturerSpecificMessage.nTextIdentityReferenceToESIFile,
                 Actual := stDiagnosticMessage.nTextIdentityReferenceToESIFile,
                 Message := 'Test $'ManufacturerSpecificMessage$' failed at $'Text identity reference to ESI file$'');
    AssertEquals(Expected := cstDiagnosticMessage_ManufacturerSpecificMessage.sTimeStamp,
                 Actual := stDiagnosticMessage.sTimeStamp,
                 Message := 'Test $'ManufacturerSpecificMessage$' failed at $'Timestamp$'');

    TEST_FINISHED();
END_IF
END_METHOD

METHOD PRIVATE TestWithUnspecifiedMessageMessage
VAR
    fbDiagnosticMessageParser : FB_DiagnosticMessageParser;
    aDiagnosticMessageBuffer : ARRAY[1..28] OF BYTE;
    stDiagnosticMessage : ST_DIAGNOSTICMESSAGE;

    // @TEST-FIXTURE UnspecifiedMessage
    cnDiagnosticBufferByte1_UnspecifiedMessage : BYTE := 16#01; // 0xE801 = Reserved for future use
    cnDiagnosticBufferByte2_UnspecifiedMessage : BYTE := 16#E8;
    cnDiagnosticBufferByte3_UnspecifiedMessage : BYTE := 16#FF; // 0xFFFF = Code 65535
    cnDiagnosticBufferByte4_UnspecifiedMessage : BYTE := 16#FF;
    cnDiagnosticBufferByte5_UnspecifiedMessage : BYTE := 2#0000_0001; // Global time stamp & warning message 
    cnDiagnosticBufferByte6_UnspecifiedMessage : BYTE := 16#FF; // Number of parameters = 255
    cnDiagnosticBufferByte7_UnspecifiedMessage : BYTE := 16#FF; // 0x61A8, Text id as reference to ESI file = 10#65535
    cnDiagnosticBufferByte8_UnspecifiedMessage : BYTE := 16#FF;
    cnDiagnosticBufferByte9_UnspecifiedMessage : BYTE := 16#FF; // Timestamp from DC clock, 16#FFFFFFFFFFFFFFFF = '2584-07-20-23:34:33.709551615'
    cnDiagnosticBufferByte10_UnspecifiedMessage : BYTE := 16#FF;
    cnDiagnosticBufferByte11_UnspecifiedMessage : BYTE := 16#FF;
    cnDiagnosticBufferByte12_UnspecifiedMessage : BYTE := 16#FF;
    cnDiagnosticBufferByte13_UnspecifiedMessage : BYTE := 16#FF;
    cnDiagnosticBufferByte14_UnspecifiedMessage : BYTE := 16#FF;
    cnDiagnosticBufferByte15_UnspecifiedMessage : BYTE := 16#FF;
    cnDiagnosticBufferByte16_UnspecifiedMessage : BYTE := 16#FF;
    cnDiagnosticBufferByte17_UnspecifiedMessage : BYTE := 2#0000_0010; // Param1 = Signed8
    cnDiagnosticBufferByte18_UnspecifiedMessage : BYTE := 2#0000_0000;
    cnDiagnosticBufferByte19_UnspecifiedMessage : BYTE := 2#0000_0101; // Port 5
    cnDiagnosticBufferByte20_UnspecifiedMessage : BYTE := 2#0000_0011; // Param2 = Signed16
    cnDiagnosticBufferByte21_UnspecifiedMessage : BYTE := 2#0000_0000;
    cnDiagnosticBufferByte22_UnspecifiedMessage : BYTE := 2#0100_0100; // EventCode = 10#65092
    cnDiagnosticBufferByte23_UnspecifiedMessage : BYTE := 2#1111_1110;
    cnDiagnosticBufferByte24_UnspecifiedMessage : BYTE := 2#0000_0010; // Param3 = Signed8
    cnDiagnosticBufferByte25_UnspecifiedMessage : BYTE := 2#0000_0000;
    cnDiagnosticBufferByte26_UnspecifiedMessage : BYTE := 2#1101_1111; // Qualifier: Instance=Reserved_7, Source=Master, Type=Notification, Mode=EventAppears
    cnDiagnosticBufferByte27_UnspecifiedMessage : BYTE := 2#0000_0000;
    cnDiagnosticBufferByte28_UnspecifiedMessage : BYTE := 2#0000_0000;

    canDiagnosticBuffer_UnspecifiedMessage : ARRAY[1..28] OF BYTE := [
                                                               cnDiagnosticBufferByte1_UnspecifiedMessage,
                                                               cnDiagnosticBufferByte2_UnspecifiedMessage,
                                                               cnDiagnosticBufferByte3_UnspecifiedMessage,
                                                               cnDiagnosticBufferByte4_UnspecifiedMessage,
                                                               cnDiagnosticBufferByte5_UnspecifiedMessage,
                                                               cnDiagnosticBufferByte6_UnspecifiedMessage,
                                                               cnDiagnosticBufferByte7_UnspecifiedMessage,
                                                               cnDiagnosticBufferByte8_UnspecifiedMessage,
                                                               cnDiagnosticBufferByte9_UnspecifiedMessage,
                                                               cnDiagnosticBufferByte10_UnspecifiedMessage,
                                                               cnDiagnosticBufferByte11_UnspecifiedMessage,
                                                               cnDiagnosticBufferByte12_UnspecifiedMessage,
                                                               cnDiagnosticBufferByte13_UnspecifiedMessage,
                                                               cnDiagnosticBufferByte14_UnspecifiedMessage,
                                                               cnDiagnosticBufferByte15_UnspecifiedMessage,
                                                               cnDiagnosticBufferByte16_UnspecifiedMessage,
                                                               cnDiagnosticBufferByte17_UnspecifiedMessage,
                                                               cnDiagnosticBufferByte18_UnspecifiedMessage,
                                                               cnDiagnosticBufferByte19_UnspecifiedMessage,
                                                               cnDiagnosticBufferByte20_UnspecifiedMessage,
                                                               cnDiagnosticBufferByte21_UnspecifiedMessage,
                                                               cnDiagnosticBufferByte22_UnspecifiedMessage,
                                                               cnDiagnosticBufferByte23_UnspecifiedMessage,
                                                               cnDiagnosticBufferByte24_UnspecifiedMessage,
                                                               cnDiagnosticBufferByte25_UnspecifiedMessage,
                                                               cnDiagnosticBufferByte26_UnspecifiedMessage,
                                                               cnDiagnosticBufferByte27_UnspecifiedMessage,
                                                               cnDiagnosticBufferByte28_UnspecifiedMessage];

    // @TEST-RESULT UnspecifiedMessage
    cstDiagnosticMessage_UnspecifiedMessage : ST_DIAGNOSTICMESSAGE :=
        (stDiagnosticCode := (eDiagnosticCodeType := E_DIAGNOSTICCODETYPE.Unspecified, nCode := 65535),
        stFlags := (eDiagnosisType := E_DIAGNOSISTYPE.WarningMessage, eTimeStampType := E_TIMESTAMPTYPE.Global,
                    nNumberOfParametersInDiagnosisMessage := 255),
        nTextIdentityReferenceToESIFile := 65535,
        sTimeStamp := '2584-07-20-23:34:33.709551615');
END_VAR
IF TEST_ORDERED('TestWithUnspecifiedMessageMessage') THEN
    GVL.fbDiagnosticMessageParser_Test_TestWithUnspecifiedMessageMessage := GVL.fbDiagnosticMessageParser_Test_TestWithUnspecifiedMessageMessage + 1; // Only for testing the framework. Ignore this.

    // @TEST-RUN
    fbDiagnosticMessageParser(anDiagnosticMessageBuffer := canDiagnosticBuffer_UnspecifiedMessage,
                              stDiagnosticMessage => stDiagnosticMessage);

    // @TEST-ASSERT
    AssertEquals(Expected := cstDiagnosticMessage_UnspecifiedMessage.stDiagnosticCode.eDiagnosticCodeType,
                 Actual := stDiagnosticMessage.stDiagnosticCode.eDiagnosticCodeType,
                 Message := 'Test $'UnspecifiedMessageMessage$' failed at $'Diagnostic code type$'');
    AssertEquals(Expected := cstDiagnosticMessage_UnspecifiedMessage.stDiagnosticCode.nCode,
                 Actual := stDiagnosticMessage.stDiagnosticCode.nCode,
                 Message := 'Test $'UnspecifiedMessageMessage$' failed at $'Diagnostic code$'');
    AssertEquals(Expected := cstDiagnosticMessage_UnspecifiedMessage.stFlags.eDiagnosisType,
                 Actual := stDiagnosticMessage.stFlags.eDiagnosisType,
                 Message := 'Test $'UnspecifiedMessageMessage$' failed at $'Diagnosis type$'');
    AssertEquals(Expected := cstDiagnosticMessage_UnspecifiedMessage.stFlags.eTimeStampType,
                 Actual := stDiagnosticMessage.stFlags.eTimeStampType,
                 Message := 'Test $'UnspecifiedMessageMessage$' failed at $'Timestamp type$'');
    AssertEquals(Expected := cstDiagnosticMessage_UnspecifiedMessage.stFlags.nNumberOfParametersInDiagnosisMessage,
                 Actual := stDiagnosticMessage.stFlags.nNumberOfParametersInDiagnosisMessage,
                 Message := 'Test $'UnspecifiedMessageMessage$' failed at $'Numbers of parameters in diagnosis message$'');
    AssertEquals(Expected := cstDiagnosticMessage_UnspecifiedMessage.nTextIdentityReferenceToESIFile,
                 Actual := stDiagnosticMessage.nTextIdentityReferenceToESIFile,
                 Message := 'Test $'UnspecifiedMessageMessage$' failed at $'Text identity reference to ESI file$'');
    AssertEquals(Expected := cstDiagnosticMessage_UnspecifiedMessage.sTimeStamp,
                 Actual := stDiagnosticMessage.sTimeStamp,
                 Message := 'Test $'UnspecifiedMessageMessage$' failed at $'Timestamp$'');

    TEST_FINISHED();
END_IF
END_METHOD

METHOD PRIVATE TestWithUnspecifiedMessageMessage_ParameterVariant
VAR
    fbDiagnosticMessageParser : FB_DiagnosticMessageParser;
    aDiagnosticMessageBuffer : ARRAY[1..28] OF BYTE;
    stDiagnosticMessage : ST_DIAGNOSTICMESSAGE;

    // @TEST-FIXTURE UnspecifiedMessage_ParameterVariant
    cnDiagnosticBufferByte1_UnspecifiedMessage_ParameterVariant : BYTE := 16#01; // 0xE801 = Reserved for future use
    cnDiagnosticBufferByte2_UnspecifiedMessage_ParameterVariant : BYTE := 16#E8;
    cnDiagnosticBufferByte3_UnspecifiedMessage_ParameterVariant : BYTE := 16#FF; // 0xFFFF = Code 65535
    cnDiagnosticBufferByte4_UnspecifiedMessage_ParameterVariant : BYTE := 16#FF;
    cnDiagnosticBufferByte5_UnspecifiedMessage_ParameterVariant : BYTE := 2#0000_0001; // Global time stamp & warning message 
    cnDiagnosticBufferByte6_UnspecifiedMessage_ParameterVariant : BYTE := 16#FF; // Number of parameters = 255
    cnDiagnosticBufferByte7_UnspecifiedMessage_ParameterVariant : BYTE := 16#FF; // 0x61A8, Text id as reference to ESI file = 10#65535
    cnDiagnosticBufferByte8_UnspecifiedMessage_ParameterVariant : BYTE := 16#FF;
    cnDiagnosticBufferByte9_UnspecifiedMessage_ParameterVariant : BYTE := 16#FF; // Timestamp from DC clock, 16#FFFFFFFFFFFFFFFF = '2584-07-20-23:34:33.709551615'
    cnDiagnosticBufferByte10_UnspecifiedMessage_ParameterVariant : BYTE := 16#FF;
    cnDiagnosticBufferByte11_UnspecifiedMessage_ParameterVariant : BYTE := 16#FF;
    cnDiagnosticBufferByte12_UnspecifiedMessage_ParameterVariant : BYTE := 16#FF;
    cnDiagnosticBufferByte13_UnspecifiedMessage_ParameterVariant : BYTE := 16#FF;
    cnDiagnosticBufferByte14_UnspecifiedMessage_ParameterVariant : BYTE := 16#FF;
    cnDiagnosticBufferByte15_UnspecifiedMessage_ParameterVariant : BYTE := 16#FF;
    cnDiagnosticBufferByte16_UnspecifiedMessage_ParameterVariant : BYTE := 16#FF;
    cnDiagnosticBufferByte17_UnspecifiedMessage_ParameterVariant : BYTE := 2#0000_0010; // Param1 = Signed8
    cnDiagnosticBufferByte18_UnspecifiedMessage_ParameterVariant : BYTE := 2#0000_0000;
    cnDiagnosticBufferByte19_UnspecifiedMessage_ParameterVariant : BYTE := 2#0000_0101; // Port 5
    cnDiagnosticBufferByte20_UnspecifiedMessage_ParameterVariant : BYTE := 2#0000_0100; // Param2 = Signed32
    cnDiagnosticBufferByte21_UnspecifiedMessage_ParameterVariant : BYTE := 2#0000_0000;
    cnDiagnosticBufferByte22_UnspecifiedMessage_ParameterVariant : BYTE := 2#1111_1111; // EventCode = 10#‭4294967295‬ (though will be interpreted as maximum 16 bits = 65535)
    cnDiagnosticBufferByte23_UnspecifiedMessage_ParameterVariant : BYTE := 2#1111_1111;
    cnDiagnosticBufferByte24_UnspecifiedMessage_ParameterVariant : BYTE := 2#1111_1111;
    cnDiagnosticBufferByte25_UnspecifiedMessage_ParameterVariant : BYTE := 2#1111_1111;
    cnDiagnosticBufferByte26_UnspecifiedMessage_ParameterVariant : BYTE := 2#0000_0010; // Param3 = Signed8
    cnDiagnosticBufferByte27_UnspecifiedMessage_ParameterVariant : BYTE := 2#0000_0000;
    cnDiagnosticBufferByte28_UnspecifiedMessage_ParameterVariant : BYTE := 2#1101_1111; // Qualifier: Instance=Reserved_7, Source=Master, Type=Notification, Mode=EventAppears

    canDiagnosticBuffer_UnspecifiedMessage_ParameterVariant : ARRAY[1..28] OF BYTE := [
                                                        cnDiagnosticBufferByte1_UnspecifiedMessage_ParameterVariant,
                                                        cnDiagnosticBufferByte2_UnspecifiedMessage_ParameterVariant,
                                                        cnDiagnosticBufferByte3_UnspecifiedMessage_ParameterVariant,
                                                        cnDiagnosticBufferByte4_UnspecifiedMessage_ParameterVariant,
                                                        cnDiagnosticBufferByte5_UnspecifiedMessage_ParameterVariant,
                                                        cnDiagnosticBufferByte6_UnspecifiedMessage_ParameterVariant,
                                                        cnDiagnosticBufferByte7_UnspecifiedMessage_ParameterVariant,
                                                        cnDiagnosticBufferByte8_UnspecifiedMessage_ParameterVariant,
                                                        cnDiagnosticBufferByte9_UnspecifiedMessage_ParameterVariant,
                                                        cnDiagnosticBufferByte10_UnspecifiedMessage_ParameterVariant,
                                                        cnDiagnosticBufferByte11_UnspecifiedMessage_ParameterVariant,
                                                        cnDiagnosticBufferByte12_UnspecifiedMessage_ParameterVariant,
                                                        cnDiagnosticBufferByte13_UnspecifiedMessage_ParameterVariant,
                                                        cnDiagnosticBufferByte14_UnspecifiedMessage_ParameterVariant,
                                                        cnDiagnosticBufferByte15_UnspecifiedMessage_ParameterVariant,
                                                        cnDiagnosticBufferByte16_UnspecifiedMessage_ParameterVariant,
                                                        cnDiagnosticBufferByte17_UnspecifiedMessage_ParameterVariant,
                                                        cnDiagnosticBufferByte18_UnspecifiedMessage_ParameterVariant,
                                                        cnDiagnosticBufferByte19_UnspecifiedMessage_ParameterVariant,
                                                        cnDiagnosticBufferByte20_UnspecifiedMessage_ParameterVariant,
                                                        cnDiagnosticBufferByte21_UnspecifiedMessage_ParameterVariant,
                                                        cnDiagnosticBufferByte22_UnspecifiedMessage_ParameterVariant,
                                                        cnDiagnosticBufferByte23_UnspecifiedMessage_ParameterVariant,
                                                        cnDiagnosticBufferByte24_UnspecifiedMessage_ParameterVariant,
                                                        cnDiagnosticBufferByte25_UnspecifiedMessage_ParameterVariant,
                                                        cnDiagnosticBufferByte26_UnspecifiedMessage_ParameterVariant,
                                                        cnDiagnosticBufferByte27_UnspecifiedMessage_ParameterVariant,
                                                        cnDiagnosticBufferByte28_UnspecifiedMessage_ParameterVariant];

    // @TEST-RESULT UnspecifiedMessageParameterVariant
    cstDiagnosticMessage_UnspecifiedMessage_ParameterVariant : ST_DIAGNOSTICMESSAGE :=
        (stDiagnosticCode := (eDiagnosticCodeType := E_DIAGNOSTICCODETYPE.Unspecified, nCode := 65535),
        stFlags := (eDiagnosisType := E_DIAGNOSISTYPE.WarningMessage, eTimeStampType := E_TIMESTAMPTYPE.Global,
                    nNumberOfParametersInDiagnosisMessage := 255),
        nTextIdentityReferenceToESIFile := 65535,
        sTimeStamp := '2584-07-20-23:34:33.709551615');
END_VAR
IF TEST_ORDERED('TestWithUnspecifiedMessageMessage_ParameterVariant') THEN
    GVL.fbDiagnosticMessageParser_Test_TestWithUnspecifiedMessageMessage_ParameterVariant := GVL.fbDiagnosticMessageParser_Test_TestWithUnspecifiedMessageMessage_ParameterVariant + 1; // Only for testing the framework. Ignore this.

    // @TEST-RUN
    fbDiagnosticMessageParser(anDiagnosticMessageBuffer := canDiagnosticBuffer_UnspecifiedMessage_ParameterVariant,
                              stDiagnosticMessage => stDiagnosticMessage);

    // @TEST-ASSERT
    AssertEquals(Expected := cstDiagnosticMessage_UnspecifiedMessage_ParameterVariant.stDiagnosticCode.eDiagnosticCodeType,
                 Actual := stDiagnosticMessage.stDiagnosticCode.eDiagnosticCodeType,
                 Message := 'Test $'UnspecifiedMessageMessage_ParameterVariant$' failed at $'Diagnostic code type$'');
    AssertEquals(Expected := cstDiagnosticMessage_UnspecifiedMessage_ParameterVariant.stDiagnosticCode.nCode,
                 Actual := stDiagnosticMessage.stDiagnosticCode.nCode,
                 Message := 'Test $'UnspecifiedMessageMessage_ParameterVariant$' failed at $'Diagnostic code$'');
    AssertEquals(Expected := cstDiagnosticMessage_UnspecifiedMessage_ParameterVariant.stFlags.eDiagnosisType,
                 Actual := stDiagnosticMessage.stFlags.eDiagnosisType,
                 Message := 'Test $'UnspecifiedMessageMessage_ParameterVariant$' failed at $'Diagnosis type$'');
    AssertEquals(Expected := cstDiagnosticMessage_UnspecifiedMessage_ParameterVariant.stFlags.eTimeStampType,
                 Actual := stDiagnosticMessage.stFlags.eTimeStampType,
                 Message := 'Test $'UnspecifiedMessageMessage_ParameterVariant$' failed at $'Timestamp type$'');
    AssertEquals(Expected := cstDiagnosticMessage_UnspecifiedMessage_ParameterVariant.stFlags.nNumberOfParametersInDiagnosisMessage,
                 Actual := stDiagnosticMessage.stFlags.nNumberOfParametersInDiagnosisMessage,
                 Message := 'Test $'UnspecifiedMessageMessage_ParameterVariant$' failed at $'Numbers of parameters in diagnosis message$'');
    AssertEquals(Expected := cstDiagnosticMessage_UnspecifiedMessage_ParameterVariant.nTextIdentityReferenceToESIFile,
                 Actual := stDiagnosticMessage.nTextIdentityReferenceToESIFile,
                 Message := 'Test $'UnspecifiedMessageMessage_ParameterVariant$' failed at $'Text identity reference to ESI file$'');
    AssertEquals(Expected := cstDiagnosticMessage_UnspecifiedMessage_ParameterVariant.sTimeStamp,
                 Actual := stDiagnosticMessage.sTimeStamp,
                 Message := 'Test $'UnspecifiedMessageMessage_ParameterVariant$' failed at $'Timestamp$'');

    TEST_FINISHED();
END_IF
END_METHOD

END_FUNCTION_BLOCK

// ---- POUs/FB_DiagnosticMessageParser.TcPOU
(*
    This function block parses a diagnostic message according to the ETG.1020 protocol enhancements.
    First 16 data bytes are mandatory data, the remaining 12 data bytes are optional data (parameter 1..n).
*)
FUNCTION_BLOCK FB_DiagnosticMessageParser
VAR_INPUT
    anDiagnosticMessageBuffer : ARRAY[1..28] OF BYTE;
END_VAR
VAR_OUTPUT
    stDiagnosticMessage : ST_DIAGNOSTICMESSAGE;
END_VAR
VAR
    anDiagnosticCodeBuffer : ARRAY[1..4] OF BYTE;
    anFlagsBuffer : ARRAY[1..2] OF BYTE;
    anTextIdentityBuffer : ARRAY[1..2] OF BYTE;
    anTimeStampBuffer : ARRAY[1..8] OF BYTE;
    anIOLinkParametersBuffer : ARRAY[1..12] OF BYTE;

    fbDiagnosticMessageDiagnosticCodeParser : FB_DiagnosticMessageDiagnosticCodeParser;
    fbDiagnosticMessageFlagsParser : FB_DiagnosticMessageFlagsParser;
    fbDiagnosticMessageTextIdentityParser : FB_DiagnosticMessageTextIdentityParser;
    fbDiagnosticMessageTimeStampParser : FB_DiagnosticMessageTimeStampParser;
END_VAR

// Parse diagnostic code
anDiagnosticCodeBuffer[1] := anDiagnosticMessageBuffer[1];
anDiagnosticCodeBuffer[2] := anDiagnosticMessageBuffer[2];
anDiagnosticCodeBuffer[3] := anDiagnosticMessageBuffer[3];
anDiagnosticCodeBuffer[4] := anDiagnosticMessageBuffer[4];
fbDiagnosticMessageDiagnosticCodeParser(anDiagnosticCodeBuffer := anDiagnosticCodeBuffer,
                                        stDiagnosticCode => stDiagnosticMessage.stDiagnosticCode);

// Parse flags
anFlagsBuffer[1] := anDiagnosticMessageBuffer[5];
anFlagsBuffer[2] := anDiagnosticMessageBuffer[6];
fbDiagnosticMessageFlagsParser(anFlagsBuffer := anFlagsBuffer,
                               stFlags => stDiagnosticMessage.stFlags);

// Parse text identity
anTextIdentityBuffer[1] := anDiagnosticMessageBuffer[7];
anTextIdentityBuffer[2] := anDiagnosticMessageBuffer[8];
fbDiagnosticMessageTextIdentityParser(anTextIdentityBuffer := anTextIdentityBuffer,
                                      nTextIdentity => stDiagnosticMessage.nTextIdentityReferenceToESIFile);

// Parse time stamp
anTimeStampBuffer[1] := anDiagnosticMessageBuffer[9];
anTimeStampBuffer[2] := anDiagnosticMessageBuffer[10];
anTimeStampBuffer[3] := anDiagnosticMessageBuffer[11];
anTimeStampBuffer[4] := anDiagnosticMessageBuffer[12];
anTimeStampBuffer[5] := anDiagnosticMessageBuffer[13];
anTimeStampBuffer[6] := anDiagnosticMessageBuffer[14];
anTimeStampBuffer[7] := anDiagnosticMessageBuffer[15];
anTimeStampBuffer[8] := anDiagnosticMessageBuffer[16];
fbDiagnosticMessageTimeStampParser(anTimeStampBuffer := anTimeStampBuffer,
                                   bIsLocalTime := (stDiagnosticMessage.stFlags.eTimeStampType = E_TIMESTAMPTYPE.Local),
                                   sTimeStamp => stDiagnosticMessage.sTimeStamp);

END_FUNCTION_BLOCK

// ---- POUs/FB_DiagnosticMessageTextIdentityParser.TcPOU
(*
    This function block parses a the part "text identity" of the diagnostic message according to the
    ETG.1020 protocol enhancements. This is the text identity according to the ESI-file.
*)
FUNCTION_BLOCK FB_DiagnosticMessageTextIdentityParser
VAR_INPUT
    anTextIdentityBuffer : ARRAY[1..2] OF BYTE;
END_VAR
VAR_OUTPUT
    nTextIdentity : UINT;
END_VAR

nTextIdentity := WORD_TO_UINT(F_WORDFromBytes(B1 := anTextIdentityBuffer[2], B0 := anTextIdentityBuffer[1]));

END_FUNCTION_BLOCK

// ---- POUs/F_WORDFromBytes.TcPOU
FUNCTION F_WORDFromBytes : WORD
VAR_INPUT
    B1 : BYTE;
    B0 : BYTE;
END_VAR

F_WORDFromBytes := SHL(BYTE_TO_WORD(B1),8) OR BYTE_TO_WORD(B0);

END_FUNCTION

// ---- POUs/FB_DiagnosticMessageTimeStampParser.TcPOU
(*
    This function block parses the timestamp. It's either the time stamp from the DC unit or the local time
    stamp (defined as the start time of the task). The time will be the local time of DCs are not supported
    or DC are only supported in 32 bit mode.
    Reference: ETG.1020.
*)
FUNCTION_BLOCK FB_DiagnosticMessageTimeStampParser
VAR_INPUT
    anTimeStampBuffer : ARRAY[1..8] OF BYTE;
    bIsLocalTime : BOOL;
END_VAR
VAR_OUTPUT
    sTimeStamp : STRING(29);
END_VAR
VAR
    nDCTime64 : LWORD;
    nDCTime64HighPart : DWORD;
    nDCTime64LowPart : DWORD;
END_VAR

nDCTime64HighPart := F_DWORDFromBytes(B3 := anTimeStampBuffer[8], B2 := anTimeStampBuffer[7],
                                      B1 := anTimeStampBuffer[6], B0 := anTimeStampBuffer[5]);
nDCTime64LowPart := F_DWORDFromBytes(B3 := anTimeStampBuffer[4], B2 := anTimeStampBuffer[3],
                                     B1 := anTimeStampBuffer[2], B0 := anTimeStampBuffer[1]);
nDCTime64 := SHL(DWORD_TO_LWORD(nDCTime64HighPart), 32) OR nDCTime64LowPart;

IF nDCTime64 = 0 THEN
    nDCTime64 := F_GetCurDcTaskTime64();
END_IF

sTimeStamp := DCTIME64_TO_STRING(in := nDCTime64);

END_FUNCTION_BLOCK

// ---- Test/FB_DiagnosticMessageTextIdentityParser_Test.TcPOU
FUNCTION_BLOCK FB_DiagnosticMessageTextIdentityParser_Test EXTENDS TcUnit.FB_TestSuite

(* The tests are run in the order that they are called. Asserts are not evaluated before the previous test has called TEST_FINISHED() *)
WhenTextIdentityLowExpectTextIdentity0();
WhenTextIdentityHighExpectTextIdentity65535();
WhenTextIdentityMedExpectTextIdentity34500();

METHOD PRIVATE WhenTextIdentityHighExpectTextIdentity65535
VAR
    fbDiagnosticMessageTextIdentityParser : FB_DiagnosticMessageTextIdentityParser;
    nTextIdentity : UINT;

    // @TEST-FIXTURE TextIdentity#High
    cnTextIdentityBufferByte1_IdentityHigh : BYTE := 16#FF; // 0xFFFF = 65535
    cnTextIdentityBufferByte2_IdentityHigh : BYTE := 16#FF;
    canTextIdentityBuffer_IdentityHigh : ARRAY[1..2] OF BYTE := [cnTextIdentityBufferByte1_IdentityHigh,
                                                                 cnTextIdentityBufferByte2_IdentityHigh];
    // @TEST-RESULT TextIdentity#High
    cnTextIdentity_IdentityHigh : UINT := 65535;
END_VAR
IF TEST_ORDERED('WhenTextIdentityHighExpectTextIdentity65535') THEN
    GVL.fbDiagnosticMessageTextIdentityParser_Test_WhenTextIdentityHighExpectTextIdentity65535 := GVL.fbDiagnosticMessageTextIdentityParser_Test_WhenTextIdentityHighExpectTextIdentity65535 + 1; // Only for testing the framework. Ignore this.

    // @TEST-RUN
    fbDiagnosticMessageTextIdentityParser(anTextIdentityBuffer := canTextIdentityBuffer_IdentityHigh,
                                          nTextIdentity => nTextIdentity);
    // @TEST-ASSERT
    AssertEquals(Expected := cnTextIdentity_IdentityHigh,
                 Actual := nTextIdentity,
                 Message := 'Test $'TextIdentity#High$' failed');

    TEST_FINISHED();
END_IF
END_METHOD

METHOD PRIVATE WhenTextIdentityLowExpectTextIdentity0
VAR
    fbDiagnosticMessageTextIdentityParser : FB_DiagnosticMessageTextIdentityParser;
    nTextIdentity : UINT;

    // @TEST-FIXTURE TextIdentity#Low
    cnTextIdentityBufferByte1_IdentityLow : BYTE := 16#00; // 0 = no text identity
    cnTextIdentityBufferByte2_IdentityLow : BYTE := 16#00;
    canTextIdentityBuffer_IdentityLow : ARRAY[1..2] OF BYTE := [cnTextIdentityBufferByte1_IdentityLow,
                                                                cnTextIdentityBufferByte2_IdentityLow];
    // @TEST-RESULT TextIdentity#Low
    cnTextIdentity_IdentityLow : UINT := 0;
END_VAR
IF TEST_ORDERED('WhenTextIdentityLowExpectTextIdentity0') THEN
    GVL.fbDiagnosticMessageTextIdentityParser_Test_WhenTextIdentityLowExpectTextIdentity0 := GVL.fbDiagnosticMessageTextIdentityParser_Test_WhenTextIdentityLowExpectTextIdentity0 + 1; // Only for testing the framework. Ignore this.

    // @TEST-RUN
    fbDiagnosticMessageTextIdentityParser(anTextIdentityBuffer := canTextIdentityBuffer_IdentityLow,
                                          nTextIdentity => nTextIdentity);
    // @TEST-ASSERT
    AssertEquals(Expected := cnTextIdentity_IdentityLow,
                 Actual := nTextIdentity,
                Message := 'Test $'TextIdentity#Low$' failed');

    TEST_FINISHED();
END_IF
END_METHOD

METHOD PRIVATE WhenTextIdentityMedExpectTextIdentity34500
VAR
    fbDiagnosticMessageTextIdentityParser : FB_DiagnosticMessageTextIdentityParser;
    nTextIdentity : UINT;

    // @TEST-FIXTURE TextIdentity#Med
    cnTextIdentityBufferByte1_IdentityMed : BYTE := 16#C4; // 0x86C4 = 34500
    cnTextIdentityBufferByte2_IdentityMed : BYTE := 16#86;
    canTextIdentityBuffer_IdentityMed : ARRAY[1..2] OF BYTE := [cnTextIdentityBufferByte1_IdentityMed,
                                                                cnTextIdentityBufferByte2_IdentityMed];
    // @TEST-RESULT TextIdentity#Med
    cnTextIdentity_IdentityMed : UINT := 34500;
END_VAR
IF TEST_ORDERED('WhenTextIdentityMedExpectTextIdentity34500') THEN
    GVL.fbDiagnosticMessageTextIdentityParser_Test_WhenTextIdentityMedExpectTextIdentity34500 := GVL.fbDiagnosticMessageTextIdentityParser_Test_WhenTextIdentityMedExpectTextIdentity34500 + 1; // Only for testing the framework. Ignore this.

    // @TEST-RUN
    fbDiagnosticMessageTextIdentityParser(anTextIdentityBuffer := canTextIdentityBuffer_IdentityMed,
                                          nTextIdentity => nTextIdentity);
    // @TEST-ASSERT
    AssertEquals(Expected := cnTextIdentity_IdentityMed,
                 Actual := nTextIdentity,
                 Message := 'Test $'TextIdentity#Med$' failed');

    TEST_FINISHED();
END_IF
END_METHOD

END_FUNCTION_BLOCK

// ---- Test/FB_DiagnosticMessageTimeStampParser_Test.TcPOU
FUNCTION_BLOCK FB_DiagnosticMessageTimeStampParser_Test EXTENDS TcUnit.FB_TestSuite

(* The tests are run in the order that they are called. Asserts are not evaluated before the previous test has called TEST_FINISHED() *)
TestWithTimestampZeroTimeExpectCurrentTime();
TestWithValidTimestampExpectSameTimestamp();

METHOD PRIVATE TestWithTimestampZeroTimeExpectCurrentTime
VAR
    fbDiagnosticMessageTimeStampParser : FB_DiagnosticMessageTimeStampParser;
    sTimeStamp : STRING(29);

    nCurrentDcTaskTime : Tc2_EtherCAT.T_DCTIME64;
    sCurrentDcTaskTimeString : STRING(29);

    // @TEST-FIXTURE time stamp zero time
    canTimeStampBuffer_TimeStampZeroTime : ARRAY[1..8] OF BYTE := [8(16#00)];
END_VAR
IF TEST_ORDERED('TestWithTimestampZeroTimeExpectCurrentTime') THEN
    GVL.fbDiagnosticMessageTimeStampParser_Test_TestWithTimestampZeroTimeExpectCurrentTime := GVL.fbDiagnosticMessageTimeStampParser_Test_TestWithTimestampZeroTimeExpectCurrentTime + 1; // Only for testing the framework. Ignore this.

    // @TEST-RUN
    fbDiagnosticMessageTimeStampParser(anTimeStampBuffer := canTimeStampBuffer_TimeStampZeroTime,
                                       sTimeStamp => sTimeStamp);
    nCurrentDcTaskTime := Tc2_EtherCAT.F_GetCurDcTaskTime64();
    sCurrentDcTaskTimeString := DCTIME64_TO_STRING(in := nCurrentDcTaskTime);

    // @TEST-ASSERT
    AssertEquals(Expected := sCurrentDcTaskTimeString,
                 Actual := sTimeStamp,
                 Message := 'Test $'TimeStamp zero time$' failed');

    TEST_FINISHED();
END_IF
END_METHOD

METHOD PRIVATE TestWithValidTimestampExpectSameTimestamp
VAR
    fbDiagnosticMessageTimeStampParser : FB_DiagnosticMessageTimeStampParser;
    sTimeStamp : STRING(29);

    // @TEST-FIXTURE TimeStamp valid time
    cnTimeStampBufferByte1_TimeStampValidTime : BYTE := 16#C0; // 0x07C76560A71025C0 = '2017-10-05-14:15:44.425035200'
    cnTimeStampBufferByte2_TimeStampValidTime : BYTE := 16#25;
    cnTimeStampBufferByte3_TimeStampValidTime : BYTE := 16#10;
    cnTimeStampBufferByte4_TimeStampValidTime : BYTE := 16#A7;
    cnTimeStampBufferByte5_TimeStampValidTime : BYTE := 16#60;
    cnTimeStampBufferByte6_TimeStampValidTime : BYTE := 16#65;
    cnTimeStampBufferByte7_TimeStampValidTime : BYTE := 16#C7;
    cnTimeStampBufferByte8_TimeStampValidTime : BYTE := 16#07;
    canTimeStampBuffer_TimeStampValidTime : ARRAY[1..8] OF BYTE := [cnTimeStampBufferByte1_TimeStampValidTime,
                                                                    cnTimeStampBufferByte2_TimeStampValidTime,
                                                                    cnTimeStampBufferByte3_TimeStampValidTime,
                                                                    cnTimeStampBufferByte4_TimeStampValidTime,
                                                                    cnTimeStampBufferByte5_TimeStampValidTime,
                                                                    cnTimeStampBufferByte6_TimeStampValidTime,
                                                                    cnTimeStampBufferByte7_TimeStampValidTime,
                                                                    cnTimeStampBufferByte8_TimeStampValidTime];
    // @TEST-RESULT TimeStamp valid time
    csTimeStamp_TimeStampValidTime : STRING(29) := '2017-10-05-14:15:44.425035200'; // T_DCTime64 = 16#07C76560A71025C0
END_VAR
IF TEST_ORDERED('TestWithValidTimestampExpectSameTimestamp') THEN
    GVL.fbDiagnosticMessageTimeStampParser_Test_TestWithValidTimestampExpectSameTimestamp := GVL.fbDiagnosticMessageTimeStampParser_Test_TestWithValidTimestampExpectSameTimestamp + 1; // Only for testing the framework. Ignore this.

    // @TEST-RUN
    fbDiagnosticMessageTimeStampParser(anTimeStampBuffer := canTimeStampBuffer_TimeStampValidTime,
                                       sTimeStamp => sTimeStamp);

    // @TEST-ASSERT
    AssertEquals(Expected := csTimeStamp_TimeStampValidTime,
                 Actual := sTimeStamp,
                 Message := 'Test $'TimeStamp zero time$' failed');

    TEST_FINISHED();
END_IF
END_METHOD

END_FUNCTION_BLOCK
